/// Axis move modulo parameter strucure
TYPE ST_AxisMoveModParameter EXTENDS ST_AxisMoveParameter :
STRUCT
	fPosition: LREAL;
	eDirection: TC2_MC2.MC_Direction;
END_STRUCT
END_TYPE

(* stored: Version 1.1.0.1, ProductVersion 3.1.4024.4
   DUT ST_AxisMoveModParameter: Id {3b1e6fa5-741a-4d97-9d3b-2a3e2c900778} *)
